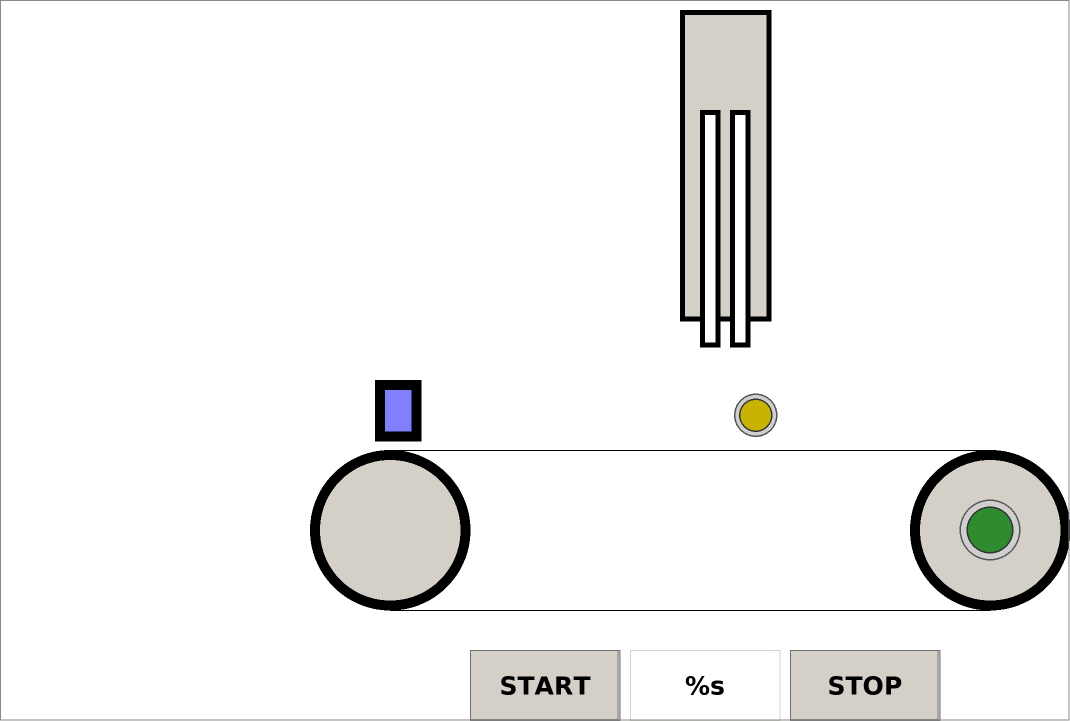
VISUALIZATION Visu  // 1070x721
    Rectangle (680,10 91x311), colour toggle: GVL.bCorking
        p2738717112: (TO_REAL(GVL.bCorking) * 50.0)
    Ellipse (310,450 160x160)
    Line (390,450) (990,450)
    Ellipse (910,450 160x160)
    Line (390,610) (990,610)
    Lamp1 (955,495 70x70), variable: GVL.bConveyor, style: Lamp-Lamp1-Green
    Rectangle (700,110 20x237), colour toggle: GVL.bWater
    Rectangle (730,110 20x237), colour toggle: GVL.bMint
    Button (470,650 150x71), "START"
        tap GVL.bStart
    Button (790,650 150x71), "STOP"
        tap GVL.bStop
    Textfield (630,650 150x71), "%s", text variable: MAIN.fbStateMachine.nStep
    Lamp1 (730,390 51x50), variable: GVL.bBottle, style: Lamp-Lamp1-Yellow
    RoundedRectangle (375,380 46x61)
        p3560616238: MAIN.fbVisuSim.fPos * 5.0
END_VISUALIZATION

(* stored: Version 1.1.0.1, ProductVersion 3.1.4024.12
   Visu Visu: Id {79eb8f98-2db4-4b83-985c-94485c8e1a1b} *)
